PROGRAM RESET_SEQ
VAR_INPUT
	Reset_seq	: INT;
	log_reset	: STRING[255];
END_VAR
VAR
	RstTON		: TON;
	RstToff		: TON;
	bOn			: BOOL;
	bLastOn		: BOOL;
	Bit1		: INT;
	Bit2		: INT;
END_VAR


	//Off time
	RstTON(IN:= NOT RstTOff.Q, PT:= T#0.2S, Q=> bOn , ET=> );
	//On time
	RstTOff(IN:= bOn, PT:= T#0.5S, Q=> , ET=> );
	
	IF bOn <> bLastOn THEN
		IF bON THEN
			IF Reset_seq < 14 THEN
				IF Reset_seq =2 THEN
					IF KR1.bInBit[1,6] AND KR2.bInBit[1,6] AND KR3.bInBit[1,6] AND KR4.bInBit[1,6] AND KR5.bInBit[1,6] THEN
						Reset_seq := Reset_seq + 1;	
					END_IF
				ELSE	
					Reset_seq := Reset_seq + 1;
				END_IF			
			ELSE
				Reset_seq 	:=0;
				bOn 		:= FALSE;
			END_IF
		END_IF
	END_IF
	
	CASE Reset_seq OF
		0:
			IF NOT GVL.KR1_bypass THEN
				FOR Bit1 := 1 TO 30 BY 1 DO
					FOR Bit2 := 0 TO 7 BY 1 DO
						KR1.bOutBit[Bit1,Bit2] := FALSE;
					END_FOR
				END_FOR
			END_IF
			IF NOT GVL.KR2_bypass THEN
				FOR Bit1 := 1 TO 8 BY 1 DO
					FOR Bit2 := 0 TO 7 BY 1 DO
						KR2.bOutBit[Bit1,Bit2] := FALSE;
					END_FOR
				END_FOR
			END_IF
			IF NOT GVL.KR3_bypass THEN
				FOR Bit1 := 1 TO 3 BY 1 DO
					FOR Bit2 := 0 TO 7 BY 1 DO
						KR3.bOutBit[Bit1,Bit2] := FALSE;
					END_FOR
				END_FOR
			END_IF
			IF NOT GVL.KR4_bypass THEN
				FOR Bit1 := 1 TO 3 BY 1 DO
					FOR Bit2 := 0 TO 7 BY 1 DO
						KR4.bOutBit[Bit1,Bit2] := FALSE;
					END_FOR
				END_FOR
			END_IF
			IF NOT GVL.KR5_bypass THEN
				FOR Bit1 := 1 TO 6 BY 1 DO
					FOR Bit2 := 0 TO 7 BY 1 DO
						KR5.bOutBit[Bit1,Bit2] := FALSE;
					END_FOR
				END_FOR
			END_IF
		1:
			IF NOT GVL.KR1_bypass THEN
				KR1.bOutBit[1,0]:=KR1.bOutBit[1,1]:=KR1.bOutBit[1,2]:=TRUE;
			END_IF
			IF NOT GVL.KR2_bypass THEN
				KR2.bOutBit[1,0]:=KR2.bOutBit[1,1]:=KR2.bOutBit[1,2]:=TRUE;
			END_IF
			IF NOT GVL.KR3_bypass THEN
				KR3.bOutBit[1,0]:=KR3.bOutBit[1,1]:=KR3.bOutBit[1,2]:=TRUE;
			END_IF
			IF NOT GVL.KR4_bypass THEN
				KR4.bOutBit[1,0]:=KR4.bOutBit[1,1]:=KR4.bOutBit[1,2]:=TRUE;
			END_IF
			IF NOT GVL.KR5_bypass THEN
				KR5.bOutBit[1,0]:=KR5.bOutBit[1,1]:=KR5.bOutBit[1,2]:=TRUE;
			END_IF
		2:
			IF NOT GVL.KR1_bypass THEN
				KR1.bOutBit[1,4] := TRUE; //1031
			END_IF
			IF NOT GVL.KR2_bypass THEN
				KR2.bOutBit[1,4] := TRUE; //1031
			END_IF
			IF NOT GVL.KR3_bypass THEN
				KR3.bOutBit[1,4] := TRUE; //1031
			END_IF
			IF NOT GVL.KR4_bypass THEN
				KR4.bOutBit[1,4] := TRUE; //1031
			END_IF
			IF NOT GVL.KR5_bypass THEN
				KR5.bOutBit[1,4] := TRUE; //1031
			END_IF
		3:
			IF NOT GVL.KR1_bypass THEN
				KR1.bOutBit[1,4] := FALSE; //1031
			END_IF
			IF NOT GVL.KR2_bypass THEN
				KR2.bOutBit[1,4] := FALSE; //1031
			END_IF
			IF NOT GVL.KR3_bypass THEN
				KR3.bOutBit[1,4] := FALSE; //1031
			END_IF
			IF NOT GVL.KR4_bypass THEN
				KR4.bOutBit[1,4] := FALSE; //1031
			END_IF
			IF NOT GVL.KR5_bypass THEN
				KR5.bOutBit[1,4] := FALSE; //1031
			END_IF
		4:
			KR1.bOutBit[1,5] := TRUE; //1032
		5:
			KR2.bOutBit[1,6] := TRUE; //1033
		6:
			KR3.bOutBit[1,5] := TRUE; //1032
		7:	
			KR4.bOutBit[1,5] := TRUE; //1032
		8:		
			KR5.bOutBit[1,5] := TRUE; //1032
		9:
			KR1.bOutBit[1,5] := FALSE; //1032
			KR1.bOutBit[1,3] := TRUE; //1030
		10:
			KR2.bOutBit[1,6] := FALSE; //1033
			KR2.bOutBit[1,3] := TRUE; //1030
		11:
			KR3.bOutBit[1,5] := FALSE; //1032
			KR3.bOutBit[1,3] := TRUE; //1030
		12:
			KR4.bOutBit[1,5] := FALSE; //1032
			KR4.bOutBit[1,3] := TRUE; //1030
		13:
			KR5.bOutBit[1,5] := FALSE; //1032
			KR5.bOutBit[1,3] := TRUE; //1030
		14:
			AUTO_MODE.Halt_Production := FALSE;
			Reset_seq :=0;
			MAIN.Reset_State := FALSE;
			MAIN.btn_Reset := FALSE;
	END_CASE
	bLastOn := bOn;

END_PROGRAM

(* stored: Version 1.1.0.1, ProductVersion 3.1.4024.12
   POU RESET_SEQ: Id {1966923e-a7dd-4db7-aeb8-7c797607c441}, SpecialFunc None *)
